ABB RAPID module: Module1.mod

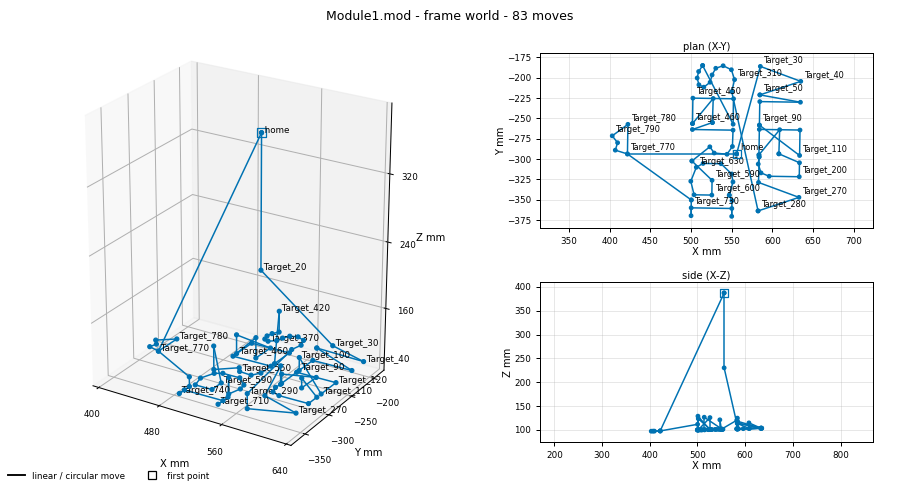
[picture p0: tool path of Module1.mod in frame world, 83 of 83 moves have a stored position in this frame; points joined in program order, loops and branches not executed]
MODULE Module1
        CONST robtarget Target_20:=[[-95.190992319,105.897899551,-128.645194861],[0.712565341,-0.009697072,0.00954606,0.701473788],[-1,-2,0,1],[9E+09,9E+09,9E+09,9E+09,9E+09,9E+09]];
    CONST robtarget Target_30:=[[-203.287806475,81.880340222,-0.000139357],[0.712565391,-0.00969701,0.009546068,0.701473738],[-1,-1,0,1],[9E+09,9E+09,9E+09,9E+09,9E+09,9E+09]];
    CONST robtarget Target_10:=[[612.211,47.138,103.585],[0,0,1,0],[0,2,-3,0],[9E+09,9E+09,9E+09,9E+09,9E+09,9E+09]];
    CONST robtarget Target_50:=[[-168.259503961,81.557373306,-11.846342015],[0.712565391,-0.00969701,0.009546068,0.701473738],[-1,-1,0,1],[9E+09,9E+09,9E+09,9E+09,9E+09,9E+09]];
    CONST robtarget home:=[[-95.190928869,101.623573364,-285.662096499],[0.712565359,-0.009697036,0.009546087,0.701473769],[-1,-2,1,1],[9E+09,9E+09,9E+09,9E+09,9E+09,9E+09]];
    CONST robtarget Target_40:=[[-185.702707204,31.879834502,0.000481612],[0.712565391,-0.00969701,0.009546068,0.701473738],[-1,-1,0,1],[9E+09,9E+09,9E+09,9E+09,9E+09,9E+09]];
    CONST robtarget Target_60:=[[-168.259518782,81.557365254,-11.846296478],[0.712565413,-0.009697022,0.009546095,0.701473714],[-1,-1,0,1],[9E+09,9E+09,9E+09,9E+09,9E+09,9E+09]];
    CONST robtarget Target_70:=[[-160.013545968,31.879850272,0.000481192],[0.712565391,-0.00969701,0.009546068,0.701473738],[-1,-1,0,1],[9E+09,9E+09,9E+09,9E+09,9E+09,9E+09]];
    CONST robtarget Target_80:=[[-160.01347919,81.880498584,-0.000143653],[0.712565391,-0.00969701,0.009546068,0.701473738],[-1,-1,0,1],[9E+09,9E+09,9E+09,9E+09,9E+09,9E+09]];
    CONST robtarget Target_90:=[[-131.04292164,81.880039418,-0.000131143],[0.712565391,-0.00969701,0.009546068,0.701473738],[-1,-1,0,1],[9E+09,9E+09,9E+09,9E+09,9E+09,9E+09]];
    CONST robtarget Target_110:=[[-94.535491408,31.879700264,0.000485298],[0.712565391,-0.00969701,0.009546068,0.701473738],[-1,-1,0,1],[9E+09,9E+09,9E+09,9E+09,9E+09,9E+09]];
    CONST robtarget Target_120:=[[-125.816329449,31.880400592,0.000466223],[0.712565391,-0.00969701,0.009546068,0.701473738],[-1,-1,0,1],[9E+09,9E+09,9E+09,9E+09,9E+09,9E+09]];
    CONST robtarget Target_130:=[[-125.816278357,81.880049398,-0.000131413],[0.712565391,-0.00969701,0.009546068,0.701473738],[-1,-1,0,1],[9E+09,9E+09,9E+09,9E+09,9E+09,9E+09]];
    CONST robtarget Target_140:=[[-94.535440317,81.879349069,-0.000112338],[0.712565391,-0.00969701,0.009546068,0.701473738],[-1,-1,0,1],[9E+09,9E+09,9E+09,9E+09,9E+09,9E+09]];
    CONST robtarget Target_150:=[[-94.535437934,81.569763928,-11.373178305],[0.712565368,-0.009697019,0.00954608,0.70147376],[-1,-1,0,1],[9E+09,9E+09,9E+09,9E+09,9E+09,9E+09]];
    CONST robtarget Target_160:=[[-125.816311746,56.879725242,0.000181009],[0.712565391,-0.00969701,0.009546068,0.701473738],[-1,-1,0,1],[9E+09,9E+09,9E+09,9E+09,9E+09,9E+09]];
    CONST robtarget Target_170:=[[-96.196409185,57.40633053,-0.000149159],[0.712565391,-0.00969701,0.009546068,0.701473738],[-1,-1,0,1],[9E+09,9E+09,9E+09,9E+09,9E+09,9E+09]];
    CONST robtarget Target_180:=[[-96.196417904,57.082797054,-11.885106772],[0.712565399,-0.009697044,0.009546092,0.701473728],[-1,-1,0,1],[9E+09,9E+09,9E+09,9E+09,9E+09,9E+09]];
    CONST robtarget Target_190:=[[-85.62139196,31.879865317,0.000480808],[0.712565391,-0.00969701,0.009546068,0.701473738],[-1,-1,0,1],[9E+09,9E+09,9E+09,9E+09,9E+09,9E+09]];
    CONST robtarget Target_200:=[[-68.40127512,31.87973448,0.000484376],[0.712565391,-0.00969701,0.009546068,0.701473738],[-1,-1,0,1],[9E+09,9E+09,9E+09,9E+09,9E+09,9E+09]];
    CONST robtarget Target_210:=[[-68.401179297,68.872964408,-0.000180801],[0.712565391,-0.00969701,0.009546068,0.701473738],[-1,-1,0,1],[9E+09,9E+09,9E+09,9E+09,9E+09,9E+09]];
    CONST robtarget Target_220:=[[-72.411824363,79.002885782,0.000162492],[0.712565391,-0.00969701,0.009546068,0.701473738],[-1,-1,0,1],[9E+09,9E+09,9E+09,9E+09,9E+09,9E+09]];
    CONST robtarget Target_230:=[[-83.190234241,82.568724181,0.000128384],[0.712565391,-0.00969701,0.009546068,0.701473738],[-1,-1,0,1],[9E+09,9E+09,9E+09,9E+09,9E+09,9E+09]];
    CONST robtarget Target_240:=[[-92.023577517,81.59582524,0.000603218],[0.712565391,-0.00969701,0.009546068,0.701473738],[-1,-1,0,1],[9E+09,9E+09,9E+09,9E+09,9E+09,9E+09]];
    CONST robtarget Target_250:=[[-92.023575369,80.982513017,-22.52911956],[0.71256538,-0.00969704,0.00954607,0.701473748],[-1,-1,0,1],[9E+09,9E+09,9E+09,9E+09,9E+09,9E+09]];
    CONST robtarget Target_260:=[[-60.621267409,81.879339615,-0.000112068],[0.712565391,-0.00969701,0.009546068,0.701473738],[-1,-1,0,1],[9E+09,9E+09,9E+09,9E+09,9E+09,9E+09]];
    CONST robtarget Target_270:=[[-43.036152452,31.879833401,0.000481692],[0.712565391,-0.00969701,0.009546068,0.701473738],[-1,-2,0,1],[9E+09,9E+09,9E+09,9E+09,9E+09,9E+09]];
    CONST robtarget Target_280:=[[-25.592949212,81.879852505,-0.000126018],[0.712565391,-0.00969701,0.009546068,0.701473738],[-1,-1,0,1],[9E+09,9E+09,9E+09,9E+09,9E+09,9E+09]];
    CONST robtarget Target_290:=[[-25.592947158,81.390270488,-17.983633705],[0.712565421,-0.009697024,0.009546137,0.701473705],[-1,-2,0,1],[9E+09,9E+09,9E+09,9E+09,9E+09,9E+09]];
    CONST robtarget Target_300:=[[-171.683200792,116.553678515,0.00032511],[0.712565391,-0.00969701,0.009546068,0.701473738],[-1,-1,0,1],[9E+09,9E+09,9E+09,9E+09,9E+09,9E+09]];
    CONST robtarget Target_310:=[[-186.552858325,113.312344405,0.000528816],[0.712565391,-0.00969701,0.009546068,0.701473738],[-1,-1,0,1],[9E+09,9E+09,9E+09,9E+09,9E+09,9E+09]];
    CONST robtarget Target_320:=[[-198.627856298,117.42479537,0.000620257],[0.712565391,-0.00969701,0.009546068,0.701473738],[-1,-1,0,1],[9E+09,9E+09,9E+09,9E+09,9E+09,9E+09]];
    CONST robtarget Target_330:=[[-203.368642756,127.615182687,0.000317903],[0.712565391,-0.00969701,0.009546068,0.701473738],[-1,-1,0,1],[9E+09,9E+09,9E+09,9E+09,9E+09,9E+09]];
    CONST robtarget Target_340:=[[-200.126555451,136.650785041,0.000439878],[0.712565391,-0.00969701,0.009546068,0.701473738],[-1,-1,0,1],[9E+09,9E+09,9E+09,9E+09,9E+09,9E+09]];
    CONST robtarget Target_350:=[[-191.861282389,141.067302014,0.000256937],[0.712565391,-0.00969701,0.009546068,0.701473738],[-1,-1,0,1],[9E+09,9E+09,9E+09,9E+09,9E+09,9E+09]];
    CONST robtarget Target_360:=[[-182.825584178,143.336685804,0.000502243],[0.712565391,-0.00969701,0.009546068,0.701473738],[-1,-1,0,1],[9E+09,9E+09,9E+09,9E+09,9E+09,9E+09]];
    CONST robtarget Target_370:=[[-176.666737699,150.994839556,0.000107352],[0.712565391,-0.00969701,0.009546068,0.701473738],[-1,-1,0,1],[9E+09,9E+09,9E+09,9E+09,9E+09,9E+09]];
    CONST robtarget Target_380:=[[-179.483101023,157.052012461,0.00027878],[0.712565391,-0.00969701,0.009546068,0.701473738],[-1,-1,0,1],[9E+09,9E+09,9E+09,9E+09,9E+09,9E+09]];
    CONST robtarget Target_390:=[[-187.809219815,159.341744928,-0.000029856],[0.712565391,-0.00969701,0.009546068,0.701473738],[-1,-1,0,1],[9E+09,9E+09,9E+09,9E+09,9E+09,9E+09]];
    CONST robtarget Target_400:=[[-195.811898543,157.639451452,0.000293308],[0.712565391,-0.00969701,0.009546068,0.701473738],[-1,-1,0,1],[9E+09,9E+09,9E+09,9E+09,9E+09,9E+09]];
    CONST robtarget Target_410:=[[-203.246780587,152.858726091,0.000387106],[0.712565391,-0.00969701,0.009546068,0.701473738],[-1,-1,0,1],[9E+09,9E+09,9E+09,9E+09,9E+09,9E+09]];
    CONST robtarget Target_420:=[[-203.246776848,152.142067563,-26.324742077],[0.712565406,-0.009697009,0.009546094,0.701473722],[-1,-1,0,1],[9E+09,9E+09,9E+09,9E+09,9E+09,9E+09]];
    CONST robtarget Target_430:=[[-131.691138551,114.20316502,0.000287611],[0.712565391,-0.00969701,0.009546068,0.701473738],[-1,-1,0,1],[9E+09,9E+09,9E+09,9E+09,9E+09,9E+09]];
    CONST robtarget Target_440:=[[-162.970976714,114.203849667,0.000268963],[0.712565391,-0.00969701,0.009546068,0.701473738],[-1,-1,0,1],[9E+09,9E+09,9E+09,9E+09,9E+09,9E+09]];
    CONST robtarget Target_450:=[[-162.970925623,164.203498472,-0.000328673],[0.712565391,-0.00969701,0.009546068,0.701473738],[-1,-1,0,1],[9E+09,9E+09,9E+09,9E+09,9E+09,9E+09]];
    CONST robtarget Target_460:=[[-131.691071772,164.203813332,-0.000337233],[0.712565391,-0.00969701,0.009546068,0.701473738],[-1,-1,0,1],[9E+09,9E+09,9E+09,9E+09,9E+09,9E+09]];
    CONST robtarget Target_470:=[[-131.69106491,163.564793986,-23.47470629],[0.712565409,-0.009697035,0.00954612,0.701473718],[-1,-1,0,1],[9E+09,9E+09,9E+09,9E+09,9E+09,9E+09]];
    CONST robtarget Target_480:=[[-162.970943325,139.204173823,-0.00004346],[0.712565391,-0.00969701,0.009546068,0.701473738],[-1,-1,0,1],[9E+09,9E+09,9E+09,9E+09,9E+09,9E+09]];
    CONST robtarget Target_490:=[[-133.35204064,139.730794793,-0.000374055],[0.712565391,-0.00969701,0.009546068,0.701473738],[-1,-1,0,1],[9E+09,9E+09,9E+09,9E+09,9E+09,9E+09]];
    CONST robtarget Target_500:=[[-133.352024749,139.045751387,-25.164532801],[0.712565365,-0.009697022,0.00954609,0.701473763],[-1,-1,0,1],[9E+09,9E+09,9E+09,9E+09,9E+09,9E+09]];
    CONST robtarget Target_510:=[[-124.397180847,164.203394636,-0.000325833],[0.712565391,-0.00969701,0.009546068,0.701473738],[-1,-1,0,1],[9E+09,9E+09,9E+09,9E+09,9E+09,9E+09]];
    CONST robtarget Target_520:=[[-124.397231939,114.203745831,0.000271803],[0.712565391,-0.00969701,0.009546068,0.701473738],[-1,-1,0,1],[9E+09,9E+09,9E+09,9E+09,9E+09,9E+09]];
    CONST robtarget Target_530:=[[-104.320465324,114.669041628,0.000610241],[0.712565391,-0.00969701,0.009546068,0.701473738],[-1,-1,0,1],[9E+09,9E+09,9E+09,9E+09,9E+09,9E+09]];
    CONST robtarget Target_540:=[[-94.636965196,121.193341053,0.000069899],[0.712565391,-0.00969701,0.009546068,0.701473738],[-1,-1,0,1],[9E+09,9E+09,9E+09,9E+09,9E+09,9E+09]];
    CONST robtarget Target_550:=[[-95.912959545,136.955135507,0.000157783],[0.712565391,-0.00969701,0.009546068,0.701473738],[-1,-1,0,1],[9E+09,9E+09,9E+09,9E+09,9E+09,9E+09]];
    CONST robtarget Target_560:=[[-103.489809283,142.444690762,-0.000224905],[0.712565391,-0.00969701,0.009546068,0.701473738],[-1,-1,0,1],[9E+09,9E+09,9E+09,9E+09,9E+09,9E+09]];
    CONST robtarget Target_570:=[[-85.702419587,164.203392396,-0.000325758],[0.712565391,-0.00969701,0.009546068,0.701473738],[-1,-1,0,1],[9E+09,9E+09,9E+09,9E+09,9E+09,9E+09]];
    CONST robtarget Target_580:=[[-85.702417974,163.41776899,-28.858809486],[0.712565394,-0.009697013,0.009546088,0.701473734],[-1,-1,0,1],[9E+09,9E+09,9E+09,9E+09,9E+09,9E+09]];
    CONST robtarget Target_590:=[[-62.323113883,139.041249199,0.000390264],[0.712565391,-0.00969701,0.009546068,0.701473738],[-1,-1,0,1],[9E+09,9E+09,9E+09,9E+09,9E+09,9E+09]];
    CONST robtarget Target_600:=[[-44.170876419,139.041496152,0.000383548],[0.712565391,-0.00969701,0.009546068,0.701473738],[-1,-1,0,1],[9E+09,9E+09,9E+09,9E+09,9E+09,9E+09]];
    CONST robtarget Target_610:=[[-44.170404213,160.881254408,0.000076887],[0.712565391,-0.00969701,0.009546068,0.701473738],[-1,-1,0,1],[9E+09,9E+09,9E+09,9E+09,9E+09,9E+09]];
    CONST robtarget Target_620:=[[-60.7831023,165.175978991,0.000208286],[0.712565391,-0.00969701,0.009546068,0.701473738],[-1,-1,0,1],[9E+09,9E+09,9E+09,9E+09,9E+09,9E+09]];
    CONST robtarget Target_630:=[[-78.044521155,158.652526463,-0.000274799],[0.712565391,-0.00969701,0.009546068,0.701473738],[-1,-1,0,1],[9E+09,9E+09,9E+09,9E+09,9E+09,9E+09]];
    CONST robtarget Target_640:=[[-82.886095862,150.427440708,0.000547684],[0.712565391,-0.00969701,0.009546068,0.701473738],[-1,-1,0,1],[9E+09,9E+09,9E+09,9E+09,9E+09,9E+09]];
    CONST robtarget Target_650:=[[-82.866382947,128.344235497,0.000478918],[0.712565391,-0.00969701,0.009546068,0.701473738],[-1,-1,0,1],[9E+09,9E+09,9E+09,9E+09,9E+09,9E+09]];
    CONST robtarget Target_660:=[[-70.507627866,115.094815901,0.000023807],[0.712565391,-0.00969701,0.009546068,0.701473738],[-1,-1,0,1],[9E+09,9E+09,9E+09,9E+09,9E+09,9E+09]];
    CONST robtarget Target_670:=[[-60.742386767,113.311763744,0.000544667],[0.712565391,-0.00969701,0.009546068,0.701473738],[-1,-1,0,1],[9E+09,9E+09,9E+09,9E+09,9E+09,9E+09]];
    CONST robtarget Target_680:=[[-44.373016883,117.607073377,-0.00034022],[0.712565391,-0.00969701,0.009546068,0.701473738],[-1,-1,0,1],[9E+09,9E+09,9E+09,9E+09,9E+09,9E+09]];
    CONST robtarget Target_690:=[[-44.373048207,117.064485545,-19.93241909],[0.71256538,-0.009697047,0.009546066,0.701473748],[-1,-1,0,1],[9E+09,9E+09,9E+09,9E+09,9E+09,9E+09]];
    CONST robtarget Target_700:=[[-37.768571525,114.203807571,0.000270152],[0.712565391,-0.00969701,0.009546068,0.701473738],[-1,-1,0,1],[9E+09,9E+09,9E+09,9E+09,9E+09,9E+09]];
    CONST robtarget Target_710:=[[-18.4012012,114.202993076,0.000292332],[0.712565391,-0.00969701,0.009546068,0.701473738],[-1,-1,0,1],[9E+09,9E+09,9E+09,9E+09,9E+09,9E+09]];
    CONST robtarget Target_720:=[[-28.084394267,114.20289273,0.00029506],[0.712565391,-0.00969701,0.009546068,0.701473738],[-1,-1,0,1],[9E+09,9E+09,9E+09,9E+09,9E+09,9E+09]];
    CONST robtarget Target_730:=[[-28.084327489,164.203541042,-0.000329785],[0.712565391,-0.00969701,0.009546068,0.701473738],[-1,-1,0,1],[9E+09,9E+09,9E+09,9E+09,9E+09,9E+09]];
    CONST robtarget Target_740:=[[-18.401134421,164.203641388,-0.000332513],[0.712565391,-0.00969701,0.009546068,0.701473738],[-1,-1,0,1],[9E+09,9E+09,9E+09,9E+09,9E+09,9E+09]];
    CONST robtarget Target_750:=[[-37.768520434,164.203456377,-0.000327483],[0.712565391,-0.00969701,0.009546068,0.701473738],[-1,-1,0,1],[9E+09,9E+09,9E+09,9E+09,9E+09,9E+09]];
    CONST robtarget Target_760:=[[-37.768548299,163.883386545,-11.75882274],[0.712565392,-0.009697044,0.009546127,0.701473735],[-1,-1,0,1],[9E+09,9E+09,9E+09,9E+09,9E+09,9E+09]];
    CONST robtarget Target_770:=[[-93.086183949,243.60739941,-0.000078579],[0.712565391,-0.00969701,0.009546068,0.701473738],[-1,-1,0,1],[9E+09,9E+09,9E+09,9E+09,9E+09,9E+09]];
    CONST robtarget Target_780:=[[-129.544655614,243.60832089,-0.000103677],[0.712565391,-0.00969701,0.009546068,0.701473738],[-1,-1,0,1],[9E+09,9E+09,9E+09,9E+09,9E+09,9E+09]];
    CONST robtarget Target_790:=[[-115.055098593,262.661410486,-0.000579178],[0.712565391,-0.00969701,0.009546068,0.701473738],[-1,-1,0,1],[9E+09,9E+09,9E+09,9E+09,9E+09,9E+09]];
    CONST robtarget Target_800:=[[-106.703531678,255.936082534,-0.00056861],[0.712565391,-0.00969701,0.009546068,0.701473738],[-1,-1,0,1],[9E+09,9E+09,9E+09,9E+09,9E+09,9E+09]];
    CONST robtarget Target_810:=[[-97.524963637,258.642443669,-0.000214352],[0.712565391,-0.00969701,0.009546068,0.701473738],[-1,-1,0,1],[9E+09,9E+09,9E+09,9E+09,9E+09,9E+09]];
    CONST robtarget Target_820:=[[-93.086183949,243.60739941,-0.000078579],[0.712565391,-0.00969701,0.009546068,0.701473738],[-1,-1,0,1],[9E+09,9E+09,9E+09,9E+09,9E+09,9E+09]];
    CONST robtarget Target_100:=[[-131.042946516,81.447572807,-15.886600076],[0.712565408,-0.009697037,0.009546111,0.701473719],[-1,-1,0,1],[9E+09,9E+09,9E+09,9E+09,9E+09,9E+09]];
!***********************************************************
    !
    ! M?dulo:  Module1
    !
    ! Descripción:
    !   <Introduzca la descripción aquí>
    !
    ! Autor: profe
    !
    ! Versión: 1.0
    !
    !***********************************************************


    !***********************************************************
    !
    ! Procedimiento Main
    !
    !   Este es el punto de entrada de su programa
    !
    !***********************************************************
    PROC main()
        !Add your code here
    ENDPROC
    PROC Path_10()
        MoveL home,v80,fine,MyNewTool\WObj:=Workobject_2;
        MoveL Target_20,v80,fine,MyNewTool\WObj:=Workobject_2;
        MoveL Target_30,v80,fine,MyNewTool\WObj:=Workobject_2;
        MoveL Target_40,v80,fine,MyNewTool\WObj:=Workobject_2;
        MoveL Target_50,v80,fine,MyNewTool\WObj:=Workobject_2;
        MoveL Target_60,v80,fine,MyNewTool\WObj:=Workobject_2;
        MoveL Target_70,v80,fine,MyNewTool\WObj:=Workobject_2;
        MoveL Target_80,v80,fine,MyNewTool\WObj:=Workobject_2;
        MoveL Target_90,v80,fine,MyNewTool\WObj:=Workobject_2;
        MoveL Target_100,v80,fine,MyNewTool\WObj:=Workobject_2;
        MoveL Target_110,v80,fine,MyNewTool\WObj:=Workobject_2;
        MoveL Target_120,v80,fine,MyNewTool\WObj:=Workobject_2;
        MoveL Target_130,v80,fine,MyNewTool\WObj:=Workobject_2;
        MoveL Target_140,v80,fine,MyNewTool\WObj:=Workobject_2;
        MoveL Target_150,v80,fine,MyNewTool\WObj:=Workobject_2;
        MoveL Target_160,v80,fine,MyNewTool\WObj:=Workobject_2;
        MoveL Target_170,v80,fine,MyNewTool\WObj:=Workobject_2;
        MoveL Target_180,v80,fine,MyNewTool\WObj:=Workobject_2;
        MoveL Target_190,v80,fine,MyNewTool\WObj:=Workobject_2;
        MoveL Target_200,v80,fine,MyNewTool\WObj:=Workobject_2;
        MoveL Target_210,v80,fine,MyNewTool\WObj:=Workobject_2;
        MoveL Target_220,v80,fine,MyNewTool\WObj:=Workobject_2;
        MoveL Target_230,v80,fine,MyNewTool\WObj:=Workobject_2;
        MoveL Target_240,v80,fine,MyNewTool\WObj:=Workobject_2;
        MoveL Target_250,v80,fine,MyNewTool\WObj:=Workobject_2;
        MoveL Target_260,v80,fine,MyNewTool\WObj:=Workobject_2;
        MoveL Target_270,v80,fine,MyNewTool\WObj:=Workobject_2;
        MoveL Target_280,v80,fine,MyNewTool\WObj:=Workobject_2;
        MoveL Target_290,v80,fine,MyNewTool\WObj:=Workobject_2;
        MoveL Target_300,v80,fine,MyNewTool\WObj:=Workobject_2;
        MoveL Target_310,v80,fine,MyNewTool\WObj:=Workobject_2;
        MoveL Target_320,v80,fine,MyNewTool\WObj:=Workobject_2;
        MoveL Target_330,v80,fine,MyNewTool\WObj:=Workobject_2;
        MoveL Target_340,v80,fine,MyNewTool\WObj:=Workobject_2;
        MoveL Target_350,v80,fine,MyNewTool\WObj:=Workobject_2;
        MoveL Target_360,v80,fine,MyNewTool\WObj:=Workobject_2;
        MoveL Target_370,v80,fine,MyNewTool\WObj:=Workobject_2;
        MoveL Target_380,v80,fine,MyNewTool\WObj:=Workobject_2;
        MoveL Target_390,v80,fine,MyNewTool\WObj:=Workobject_2;
        MoveL Target_400,v80,fine,MyNewTool\WObj:=Workobject_2;
        MoveL Target_410,v80,fine,MyNewTool\WObj:=Workobject_2;
        MoveL Target_420,v80,fine,MyNewTool\WObj:=Workobject_2;
        MoveL Target_430,v80,fine,MyNewTool\WObj:=Workobject_2;
        MoveL Target_440,v80,fine,MyNewTool\WObj:=Workobject_2;
        MoveL Target_450,v80,fine,MyNewTool\WObj:=Workobject_2;
        MoveL Target_460,v80,fine,MyNewTool\WObj:=Workobject_2;
        MoveL Target_470,v80,fine,MyNewTool\WObj:=Workobject_2;
        MoveL Target_480,v80,fine,MyNewTool\WObj:=Workobject_2;
        MoveL Target_490,v80,fine,MyNewTool\WObj:=Workobject_2;
        MoveL Target_500,v80,fine,MyNewTool\WObj:=Workobject_2;
        MoveL Target_510,v80,fine,MyNewTool\WObj:=Workobject_2;
        MoveL Target_520,v80,fine,MyNewTool\WObj:=Workobject_2;
        MoveL Target_530,v80,fine,MyNewTool\WObj:=Workobject_2;
        MoveL Target_540,v80,fine,MyNewTool\WObj:=Workobject_2;
        MoveL Target_550,v80,fine,MyNewTool\WObj:=Workobject_2;
        MoveL Target_560,v80,fine,MyNewTool\WObj:=Workobject_2;
        MoveL Target_570,v80,fine,MyNewTool\WObj:=Workobject_2;
        MoveL Target_580,v80,fine,MyNewTool\WObj:=Workobject_2;
        MoveL Target_590,v80,fine,MyNewTool\WObj:=Workobject_2;
        MoveL Target_600,v80,fine,MyNewTool\WObj:=Workobject_2;
        MoveL Target_610,v80,fine,MyNewTool\WObj:=Workobject_2;
        MoveL Target_620,v80,fine,MyNewTool\WObj:=Workobject_2;
        MoveL Target_630,v80,fine,MyNewTool\WObj:=Workobject_2;
        MoveL Target_640,v80,fine,MyNewTool\WObj:=Workobject_2;
        MoveL Target_650,v80,fine,MyNewTool\WObj:=Workobject_2;
        MoveL Target_660,v80,fine,MyNewTool\WObj:=Workobject_2;
        MoveL Target_670,v80,fine,MyNewTool\WObj:=Workobject_2;
        MoveL Target_680,v80,fine,MyNewTool\WObj:=Workobject_2;
        MoveL Target_690,v80,fine,MyNewTool\WObj:=Workobject_2;
        MoveL Target_700,v80,fine,MyNewTool\WObj:=Workobject_2;
        MoveL Target_710,v80,fine,MyNewTool\WObj:=Workobject_2;
        MoveL Target_720,v80,fine,MyNewTool\WObj:=Workobject_2;
        MoveL Target_730,v80,fine,MyNewTool\WObj:=Workobject_2;
        MoveL Target_740,v80,fine,MyNewTool\WObj:=Workobject_2;
        MoveL Target_750,v80,fine,MyNewTool\WObj:=Workobject_2;
        MoveL Target_760,v80,fine,MyNewTool\WObj:=Workobject_2;
        MoveL Target_770,v80,fine,MyNewTool\WObj:=Workobject_2;
        MoveL Target_780,v80,fine,MyNewTool\WObj:=Workobject_2;
        MoveL Target_790,v80,fine,MyNewTool\WObj:=Workobject_2;
        MoveL Target_800,v80,fine,MyNewTool\WObj:=Workobject_2;
        MoveL Target_810,v80,fine,MyNewTool\WObj:=Workobject_2;
        MoveL Target_820,v80,fine,MyNewTool\WObj:=Workobject_2;
        MoveL home,v1000,z100,MyNewTool\WObj:=Workobject_2;
    ENDPROC
ENDMODULE
